(* PLC project  *)

PROGRAM P
  VAR
    CTUD_0 : CTUD;
  END_VAR
  VAR  (* added by the conversion: wires and edge detectors of the diagram *)
    R_TRIG1 : R_TRIG;
    R_TRIG2 : R_TRIG;
  END_VAR

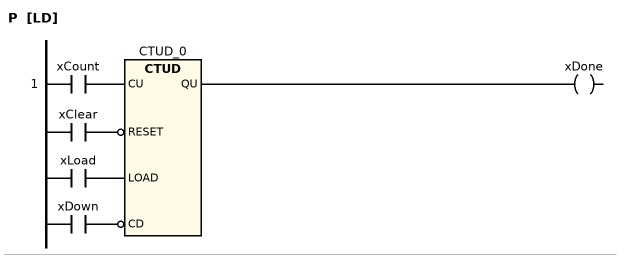
(* LD diagram, written out as Structured Text *)
R_TRIG1(CLK := xLoad);
R_TRIG2(CLK := NOT xDown);
CTUD_0(CU := xCount, RESET := NOT xClear, LOAD := R_TRIG1.Q, CD := R_TRIG2.Q);
xDone := CTUD_0.QU;
END_PROGRAM
